{attribute 'qualified_only'}
{attribute 'strict'}
{attribute 'to_string'}
TYPE TRIM_MODE :
(
	LEFT_AND_RIGHT := 0,
	LEFT,
	RIGHT
);
END_TYPE

(* stored: Version 1.1.0.1
   DUT TRIM_MODE: Id {88ff6103-4494-45b4-aac5-9792fdee98dc} *)
